Staubli VAL3: login.pgx

public program login(sio& x_sioSocket (dimensions=1), string x_sUser (dimensions=1), string x_sPassword (dimensions=1), num& x_nCamID (dimensions=1), bool& x_bError[] (dimensions=1))
  local string l_sMsg
  local bool l_bError
begin
  //-----------------------------------------------------------------------
  //Header begin
  //Description of program
  //  Login to camera via TCP/IP socket port 1023, password pair
  // (usually "admin" and "").
  //  Returns camera's ID of type num for further communication with the camera.
  //
  //Input parameters
  //  string x_sUser :
  //    role : user name
  //  string x_sPassword :
  //    role : password for the user x_sUser
  //
  //Output parameters
  //  sio x_sioSocket :
  //    role : CS8 client socket
  //  num x_nCamID :
  //    role : returns camera's ID for further operations as the lib can
  //          communicate with more that 1 camera.
  //    posssible values : - first camera (first login)  : x_nCamID=1
  //                       - second camera (second login): x_nCamID=2
  //                       - ...
  //  bool x_bError :
  //    role : returns true if an error occurred and false otherwise
  //
  //Examples
  //  call login(cognex1,"admin","",nCamID,x_bError)
  //
  //History
  //  Creation : 19-05-08 - f.Rob
  //Header end
  //-----------------------------------------------------------------------
  if bDebugProgram
    putln("Cognex login")
  endIf
  // Check available ID
  l_bError=false
  if bGetID==true
    call isIDAvailable(x_nCamID,l_bError)
  endIf
  if l_bError==false
    nProgram[x_nCamID]=1
    sioLink(cCamera[x_nCamID].sSocket,x_sioSocket)
    // Read welcome string
    call readSocket(x_nCamID,l_sMsg,x_bError)
    // Send user name
    call readLogin(x_nCamID,l_sMsg,x_bError)
    call writeSocket(x_nCamID,x_sUser)
    // Send password
    call readLogin(x_nCamID,l_sMsg,x_bError)
    call writeSocket(x_nCamID,x_sPassword)
    // Read login result
    call readSocket(x_nCamID,l_sMsg,x_bError)
    x_bError=find(l_sMsg,"User Logged In")==-1
    if x_bError
      cCamera[x_nCamID].nErrorCode=1
      cCamera[x_nCamID].bConnected=false
      if bDebugProgram
        putln("Login : failed")
      endIf
    else
      cCamera[x_nCamID].bConnected=true
    endIf
  else
    x_bError=true
    nLibErrorCode=203
  endIf
end
